FUNCTION_BLOCK RampLimitFS (* Setpoint Ramp: Step up and down Values with Fast and Slow mode *)
  (* Standard: 61499-1; Description: Copyright (c) 2024 HR Agrartechnik GmbH This program and the accompanying materials are made available under the terms of the Eclipse Public License 2.0 which is available at https://www.eclipse.org/legal/epl-2.0/ SPDX-License-Identifier: EPL-2.0 Setpoint Ramp: Step up and down Values, like well-known for the cruise control in your Car. Long press increase or decrease by 10, short press increase or decrease at 1. this FB adds Maximum and Minimum Value and also Inputs to set them. For some Applications it is neccessary to store the setpoint in Non-Volatile Storage, e.g. with a ini File, for this we have here a LOAD event input which loads value from the PV input *)
  (* Version 3.2, 2026-08-12, Franz Höpfinger, HR Agrartechnik GmbH, add upper and lower limit reached indicators *)
  (* Version 3.1, 2026-08-12, Franz Höpfinger, HR Agrartechnik GmbH, add init and correct WITH. *)
  (* Version 3.0, 2025-04-14, Patrick Aigner, changed package *)
  (* Version 1.1, 2024-10-02, Franz Höpfinger, HR Agrartechnik GmbH, Rename to RampLimitFS *)
  (* Version 1.0, 2024-09-20, Franz Höpfinger, HR Agrartechnik GmbH *)
  PACKAGE eclipse4diac::signalprocessing;
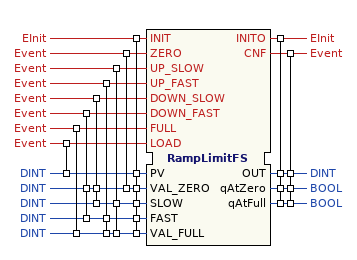
  EVENT_INPUT
    INIT : EInit WITH PV, VAL_ZERO, SLOW, FAST, VAL_FULL; (* Initialize all data inputs (PV, VAL_ZERO, SLOW, FAST, VAL_FULL) - without this, e.g. VAL_FULL is never read until FULL is fired once, breaking the UP_FAST/UP_SLOW clamp against it *)
    ZERO WITH VAL_ZERO; (* Set OUT to VAL_ZERO *)
    UP_SLOW WITH SLOW, VAL_FULL; (* Increase OUT by SLOW, clamped to VAL_FULL *)
    UP_FAST WITH FAST, VAL_FULL; (* Increase OUT by FAST, clamped to VAL_FULL *)
    DOWN_SLOW WITH SLOW, VAL_ZERO; (* Decrease OUT by SLOW, clamped to VAL_ZERO *)
    DOWN_FAST WITH FAST, VAL_ZERO; (* Decrease OUT by FAST, clamped to VAL_ZERO *)
    FULL WITH VAL_FULL; (* Set OUT to VAL_FULL *)
    LOAD WITH PV; (* Load PV into OUT *)
  END_EVENT
  EVENT_OUTPUT
    INITO : EInit WITH OUT, qAtZero, qAtFull; (* Initialization Confirmation *)
    CNF WITH OUT, qAtZero, qAtFull; (* Execution Confirmation *)
  END_EVENT
  VAR_INPUT
    PV : DINT; (* Preset Value *)
    VAL_ZERO : DINT; (* Minimum Value *)
    SLOW : DINT; (* Value for slower Change *)
    FAST : DINT; (* Value for faster change *)
    VAL_FULL : DINT; (* Maximum Value *)
  END_VAR
  VAR_OUTPUT
    OUT : DINT; (* Output *)
    qAtZero : BOOL; (* TRUE if OUT is at or below VAL_ZERO (lower limit reached) *)
    qAtFull : BOOL; (* TRUE if OUT is at or above VAL_FULL (upper limit reached) *)
  END_VAR
  EC_STATES
    INIT : INIT -> INITO;
    ZERO : ZERO -> CNF;
    UP_SLOW : UP_SLOW -> CNF;
    UP_FAST : UP_FAST -> CNF;
    DOWN_SLOW : DOWN_SLOW -> CNF;
    DOWN_FAST : DOWN_FAST -> CNF;
    FULL : FULL -> CNF;
    LOAD : LOAD -> CNF;
  END_STATES
  ALGORITHM INIT IN ST: (* Reset OUT to VAL_ZERO. Runs once at INIT, after VAL_ZERO/VAL_FULL/SLOW/FAST/PV have all been latched (see INIT event's With-list) - gives a deterministic starting OUT and guarantees VAL_FULL/VAL_ZERO are available for the first UP/DOWN clamp, instead of their DINT default of 0. *)
OUT := VAL_ZERO;
qAtZero := LE(OUT, VAL_ZERO);
qAtFull := GE(OUT, VAL_FULL);
  END_ALGORITHM
  ALGORITHM ZERO IN ST: (* Jump straight to the lower limit: OUT := VAL_ZERO. No clamping needed, VAL_ZERO is the limit itself. *)
OUT := VAL_ZERO;
qAtZero := LE(OUT, VAL_ZERO);
qAtFull := GE(OUT, VAL_FULL);
  END_ALGORITHM
  ALGORITHM UP_SLOW IN ST: (* Small step up: OUT += SLOW, then clamp down to VAL_FULL if it overshot. VAL_FULL must be latched (see this event's With-list) or the clamp uses a stale/zero value. *)
OUT := ADD(OUT, SLOW);
IF GT(OUT, VAL_FULL) THEN
	OUT := VAL_FULL;
END_IF;
qAtZero := LE(OUT, VAL_ZERO);
qAtFull := GE(OUT, VAL_FULL);
  END_ALGORITHM
  ALGORITHM UP_FAST IN ST: (* Big step up: OUT += FAST, then clamp down to VAL_FULL if it overshot. VAL_FULL must be latched (see this event's With-list) or the clamp uses a stale/zero value. *)
OUT := ADD(OUT, FAST);
IF GT(OUT, VAL_FULL) THEN
	OUT := VAL_FULL;
END_IF;
qAtZero := LE(OUT, VAL_ZERO);
qAtFull := GE(OUT, VAL_FULL);
  END_ALGORITHM
  ALGORITHM DOWN_SLOW IN ST: (* Small step down: OUT -= SLOW, then clamp up to VAL_ZERO if it undershot. VAL_ZERO must be latched (see this event's With-list) or the clamp uses a stale/zero value. *)
OUT := SUB(OUT, SLOW);
IF LT(OUT, VAL_ZERO) THEN
	OUT := VAL_ZERO;
END_IF;
qAtZero := LE(OUT, VAL_ZERO);
qAtFull := GE(OUT, VAL_FULL);
  END_ALGORITHM
  ALGORITHM DOWN_FAST IN ST: (* Big step down: OUT -= FAST, then clamp up to VAL_ZERO if it undershot. VAL_ZERO must be latched (see this event's With-list) or the clamp uses a stale/zero value. *)
OUT := SUB(OUT, FAST);
IF LT(OUT, VAL_ZERO) THEN
	OUT := VAL_ZERO;
END_IF;
qAtZero := LE(OUT, VAL_ZERO);
qAtFull := GE(OUT, VAL_FULL);
  END_ALGORITHM
  ALGORITHM FULL IN ST: (* Jump straight to the upper limit: OUT := VAL_FULL. No clamping needed, VAL_FULL is the limit itself. *)
OUT := VAL_FULL;
qAtZero := LE(OUT, VAL_ZERO);
qAtFull := GE(OUT, VAL_FULL);
  END_ALGORITHM
  ALGORITHM LOAD IN ST: (* Load an externally supplied preset directly into OUT: OUT := PV. Not clamped to VAL_ZERO/VAL_FULL - caller is expected to pass an already-valid value (e.g. a persisted setpoint restored from non-volatile storage), but qAtZero/qAtFull still reflect where it landed relative to the limits. *)
OUT := PV;
qAtZero := LE(OUT, VAL_ZERO);
qAtFull := GE(OUT, VAL_FULL);
  END_ALGORITHM
END_FUNCTION_BLOCK
